KUKA KRL program: ResetIO.src

&ACCESS RVEO
&REL 1167
&PARAM DISKPATH = KRC:\R1\Program\KUKA\Subprogs
DEF ResetIO ( )

   boRobotUnknowPos  = FALSE
   boButtonPanel     = FALSE
   biStartProgram    = FALSE
   biStopRobot       = FALSE

   OUT_LightRed      = FALSE
   OUT_LightGreen    = FALSE
   OUT_LightBlue     = FALSE
   OUT_LightYelow    = FALSE

END
